{attribute 'linkalways'} 
{attribute 'no_explicit_call' := 'This FB is a CLASS and must be accessed using methods or properties'}
{attribute 'enable_dynamic_creation'}
FUNCTION_BLOCK Node_F_VN_RotateImageExp EXTENDS VisionNode
VAR
    ipSrcImage : _ITcVnImage;
    ipDestImage : _ITcVnImage;
    fAngleDeg : _LREAL(0.0);
    bAdjustDestSize : _BOOL(FALSE);
    hrPrev : _HRESULT(S_OK);
	hresult : _HRESULT(S_OK);
END_VAR

METHOD PUBLIC  Clone : I_Node
VAR
	pNode : POINTER TO Node_F_VN_RotateImageExp;
END_VAR
pNode := __NEW(Node_F_VN_RotateImageExp);
Clone := pNode^;
END_METHOD

METHOD FB_init : BOOL
VAR_INPUT
	bInitRetains : BOOL; // if TRUE, the retain variables are initialized (warm start / cold start)
	bInCopyCode : BOOL;  // if TRUE, the instance afterwards gets moved into the copy code (online change)
END_VAR
AddInput('ipSrcImage', ipSrcImage);
AddParameter('fAngleDeg', fAngleDeg);
AddParameter('bAdjustDestSize', bAdjustDestSize);
AddInput('hrPrev', hrPrev);
AddOutput('ipDestImage', ipDestImage);
AddOutput('hresult',hresult);
END_METHOD

METHOD PROTECTED OnExecute
hresult.Value := F_VN_RotateImageExp(
    ipSrcImage := ipSrcImage.Value,
	ipDestImage := ipDestImage.Value,
    fAngleDeg := fAngleDeg.Value,
    bAdjustDestSize := bAdjustDestSize.Value,
	hrPrev:= hrPrev.Value);
END_METHOD

METHOD PUBLIC PreExecutionCheck
VAR_INPUT
	Check : I_PreExecutionChecks;
END_VAR
Check.IsTrue(ipSrcImage.IsValid, 'ipSrcImage must contain an image');
END_METHOD

END_FUNCTION_BLOCK

(* stored: Version 1.1.0.1, ProductVersion 3.1.4024.13
   POU Node_F_VN_RotateImageExp: Id {0d850de1-cb6b-0748-20b9-ae7d775db687}, SpecialFunc None
   Folder Constructor: Id {7dc36c37-1943-06d0-21fc-081c5a4f4806}
   Method Clone: Id {23fe72a2-6cb2-0d36-0c43-3ec1fd765cde}
   Method FB_init: Id {7c9620fc-071f-0bbc-28e0-a6c335bfa24b}
   Method OnExecute: Id {e5096a2f-3f69-0ca1-3da3-0f176bcffb80}
   Method PreExecutionCheck: Id {5d43fe9b-8e77-0376-1835-d1672f636b7a} *)
